Staubli VAL3: start.pgx

program start()
  local num i
  local num nBuffer[1 30]
  local num nbc[30 1]
  local num ndf[30 1 1]
  local num nt[30]
  local string sBufer
begin
  //call external:start()
  //pDest=here(tActive,frActive)
end
